PROGRAM MAIN
VAR
	
	boot :BOOL := TRUE;

	


END_VAR

IF boot THEN
	boot:=FALSE;
END_IF


MaBaseState();

GetEtherSta();

Sensor();

AutoMain();

GroupFx();

ExpConver();

AxisAction();



// SQL 專案資料讀寫功能
ReadSQLData();

LogFx();

MsgMain();

LightTower();

Button();

GetEtherSta();

ACTION init:

END_ACTION

END_PROGRAM

(* stored: Version 1.1.0.1, ProductVersion 3.1.4026.13
   POU MAIN: Id {b8aaffc0-b28a-4b26-916a-f66736143d5b}, SpecialFunc None
   Action init: Id {1f5dfe6f-0bec-44ca-887f-137cb5faa6b0} *)
